FUNCTION_BLOCK _Array0to10OfBool_TestSuite EXTENDS TcUnit.FB_TestSuite
VAR
END_VAR

TestAddress();
TestBaseDatatype();
TestClearReference();
TestClone();
TestGetElementByIndex();
TestTypeNameReturnsExpected();
TestIdentifierReturnsExpected();
TestLength();
TestLowerBound();
TestMakeReferenceToFollowsReference();
TestMakeReferenceToUpdatesReference();
TestSize();
TestSerializeTypeWith();
TestSerializeWith();
TestTryDeserializeFrom();
TestTryMakeReferenceToFollowsReference();
TestTryMakeReferenceToUpdatesReference();
TestUpperBound();
TestValueReturnsExpectedAfterChange();

METHOD PUBLIC TestAddress
VAR
    _type : _Array0to10OfBool;
    notExpected : PVOID := 0;
    actual : PVOID;
END_VAR
TEST('TestAddress');

actual := _type.Address;

AssertFalse(
    Condition := (notExpected = actual),
    Message := 'Type did not return a valid address.'
);

TEST_FINISHED();
END_METHOD

METHOD PUBLIC TestBaseDatatype
VAR
    _type : _Array0to10OfBool;
    expected : T_MAXSTRING := 'BOOL';
    actual : T_MAXSTRING;
END_VAR
TEST('TestBaseDatatype');

actual := _type.BaseDatatype.TypeName;

AssertEquals_STRING(
    Expected := expected,
    Actual := actual,
    Message := 'Type did not return the correct base type'
);

TEST_FINISHED();
END_METHOD

METHOD PUBLIC TestClearReference
VAR
    _type : _Array0to10OfBool;
	target : ARRAY [0..10] OF BOOL;
    expected : ARRAY [0..10] OF BOOL := [FALSE,FALSE,FALSE,FALSE,FALSE,FALSE,FALSE,FALSE,FALSE,FALSE,FALSE];
    actual : ARRAY [0..10] OF BOOL;
END_VAR
TEST('TestClearReference');

_type.MakeReferenceTo(target);
_type.ClearReference();
target[5] := TRUE;

actual := _type.Value;

AssertEquals(
    Expected := expected,
    Actual := actual,
    Message := 'Value incorrectly followed target change'
);

TEST_FINISHED();
END_METHOD

METHOD PUBLIC TestClone
VAR
    _type : _Array0to10OfBool;
	clone : I_Datatype;
	isValidClone : BOOL;
	compareResult : DINT;
END_VAR
TEST('TestClone');

clone := _type.Clone();

isValidClone := clone <> 0;

IF isValidClone THEN
	compareResult := memcmp(_type.Address, clone.Address, clone.Size);
END_IF

AssertTrue(
	Condition := isValidClone,
	Message := 'Clone did not produce a clone'
);

AssertEquals_DINT(
	Expected := 0,
    Actual := compareResult,
    Message := 'Clone did not return a valid clone.'
);

clone.Dispose();

TEST_FINISHED();
END_METHOD

METHOD PUBLIC TestGetElementByIndex
VAR
	_type : _Array0to10OfBool;
    expected : ARRAY [0..10] OF BOOL := [FALSE,FALSE,FALSE,FALSE,FALSE,TRUE,FALSE,FALSE,FALSE,FALSE,FALSE];
    actual : ARRAY [0..10] OF BOOL;
END_VAR
TEST('TestGetElementByIndex');

_type.GetElementByIndex(5).Value := TRUE;

actual := _type.Value;

AssertEquals(
    Expected := expected,
    Actual := actual,
    Message := 'Value did not update target'
);

TEST_FINISHED();
END_METHOD

METHOD PUBLIC TestIdentifierReturnsExpected
VAR
    _type : _Array0to10OfBool;
    expected : STRING := 'ARRAY [0..10] OF BOOL';
    actual : STRING;
END_VAR
TEST('TestIdentifierReturnsExpected');

actual := _type.Identifier;

AssertEquals_STRING(
    Expected := expected,
    Actual := actual,
    Message := 'Type did not return correct iec type.'
);

TEST_FINISHED();
END_METHOD

METHOD PUBLIC TestLength
VAR
    _type : _Array0to10OfBool;
    expected : UDINT := 11;
    actual : UDINT;
END_VAR
TEST('TestLength');

actual := _type.Length;

AssertEquals_UDINT(
    Expected := Expected,
    Actual := actual,
    Message := 'Type did not return the correct array length.'
);

TEST_FINISHED();
END_METHOD

METHOD PUBLIC TestLowerBound
VAR
    _type : _Array0to10OfBool;
    expected : DINT := 0;
    actual : DINT;
END_VAR
TEST('TestLowerBound');

actual := _type.LowerBound;

AssertEquals_DINT(
    Expected := Expected,
    Actual := actual,
    Message := 'Type did not return the correct array lower bound.'
);

TEST_FINISHED();
END_METHOD

METHOD PUBLIC TestMakeReferenceToFollowsReference
VAR
	_type : _Array0to10OfBool;
	target : ARRAY [0..10] OF BOOL;
    expected : ARRAY [0..10] OF BOOL := [TRUE,FALSE,TRUE,FALSE,TRUE,FALSE,TRUE,FALSE,TRUE,FALSE,TRUE];
    actual : ARRAY [0..10] OF BOOL;
END_VAR
TEST('TestMakeReferenceToFollowsReference');

_type.MakeReferenceTo(target);
target[0] := TRUE;
target[2] := TRUE;
target[4] := TRUE;
target[6] := TRUE;
target[8] := TRUE;
target[10] := TRUE;

actual := _type.Value;

AssertEquals(
    Expected := expected,
    Actual := actual,
    Message := 'Value did not follow target change'
);

TEST_FINISHED();
END_METHOD

METHOD PUBLIC TestMakeReferenceToUpdatesReference
VAR
	_type : _Array0to10OfBool;
	target : ARRAY [0..10] OF BOOL;
    expected : ARRAY [0..10] OF BOOL := [TRUE,FALSE,TRUE,FALSE,TRUE,FALSE,TRUE,FALSE,TRUE,FALSE,TRUE];
    actual : ARRAY [0..10] OF BOOL;
END_VAR
TEST('TestMakeReferenceToUpdatesReference');

_type.MakeReferenceTo(target);
_type.Value[0] := TRUE;
_type.Value[2] := TRUE;
_type.Value[4] := TRUE;
_type.Value[6] := TRUE;
_type.Value[8] := TRUE;
_type.Value[10] := TRUE;

actual := target;

AssertEquals(
    Expected := expected,
    Actual := actual,
    Message := 'Value did not update target'
);

TEST_FINISHED();
END_METHOD

METHOD PUBLIC TestSerializeTypeWith
VAR
    _type : _Array0to10OfBool;
    serializer : JsonSerializer;
    expected : STRING(1000) := '{"typeName":"ARRAY","identifier":"ARRAY [0..10] OF BOOL","baseType":{"typeName":"BOOL"}}';
    actual : STRING(1000);
END_VAR
TEST('TestSerializeTypeWith');

serializer.Reset();
_type.SerializeTypeWith(serializer);
serializer.TryGetSerializedData(ADR(actual), SIZEOF(actual));

AssertEquals_STRING(
    Expected := expected,
    Actual := actual,
    Message := 'Serialization of type did not return correct string.'
);

TEST_FINISHED();
END_METHOD

METHOD PUBLIC TestSerializeWith
VAR
    _type : _Array0to10OfBool;
    serializer : JsonSerializer;
    expected : STRING(500) := '[true,false,true,false,true,false,true,false,true,false,true]';
    actual : STRING(500);
END_VAR
TEST('TestSerializeWith');

_type.Value[0] := TRUE;
_type.Value[2] := TRUE;
_type.Value[4] := TRUE;
_type.Value[6] := TRUE;
_type.Value[8] := TRUE;
_type.Value[10] := TRUE;

serializer.Reset();
_type.SerializeWith(serializer);
serializer.TryGetSerializedData(ADR(actual), SIZEOF(actual));

AssertEquals_STRING(
    Expected := expected,
    Actual := actual,
    Message := 'Serialization of type data did not return correct string.'
);

TEST_FINISHED();
END_METHOD

METHOD PUBLIC TestSize
VAR
    _type : _Array0to10OfBool;
	example : ARRAY [0..10] OF BOOL;
    expected : UDINT := SIZEOF(example);
    actual : UDINT;
END_VAR
TEST('TestSize');

actual := _type.Size;

AssertEquals_UDINT(
    Expected := Expected,
    Actual := actual,
    Message := 'Type did not return the correct size.'
);

TEST_FINISHED();
END_METHOD

METHOD PUBLIC TestTryDeserializeFrom
VAR
    deserializer : JsonDeserializer;
    feedback : DeserializerFeedback;
    json : STRING(500) := '[true,false,true,false,true,false,true,false,true,false,true]';
    _type : _Array0to10OfBool;
    expected :  ARRAY [0..10] OF BOOL := [TRUE,FALSE,TRUE,FALSE,TRUE,FALSE,TRUE,FALSE,TRUE,FALSE,TRUE];
    actual : ARRAY [0..10] OF BOOL;
 END_VAR
TEST('TestTryDeserializeFrom');

deserializer.Reset();
deserializer.TryLoad(json);
_type.TryDeserializeFrom(Deserializer, Feedback);

actual := _type.Value;

AssertEquals(
    Expected := expected,
    Actual := actual,
    Message := 'Type did not deserialize correctly.'
);

TEST_FINISHED();
END_METHOD

METHOD PUBLIC TestTryMakeReferenceToFollowsReference
VAR
    _type : _Array0to10OfBool;
	target : _Array0to10OfBool;
    expected : ARRAY [0..10] OF BOOL := [TRUE,FALSE,TRUE,FALSE,TRUE,FALSE,TRUE,FALSE,TRUE,FALSE,TRUE];
    actual :  ARRAY [0..10] OF BOOL;
END_VAR
TEST('TestTryMakeReferenceToFollowsReference');

_type.TryMakeReferenceTo(target);
target.Value[0] := TRUE;
target.Value[2] := TRUE;
target.Value[4] := TRUE;
target.Value[6] := TRUE;
target.Value[8] := TRUE;
target.Value[10] := TRUE;

actual := _type.Value;

AssertEquals(
    Expected := expected,
    Actual := actual,
    Message := 'Value did not follow target change'
);

TEST_FINISHED();
END_METHOD

METHOD PUBLIC TestTryMakeReferenceToUpdatesReference
VAR
    _type : _Array0to10OfBool;
	target : _Array0to10OfBool;
    expected : ARRAY [0..10] OF BOOL := [TRUE,FALSE,TRUE,FALSE,TRUE,FALSE,TRUE,FALSE,TRUE,FALSE,TRUE];
    actual :  ARRAY [0..10] OF BOOL;
END_VAR
TEST('TestTryMakeReferenceToUpdatesReference');

_type.TryMakeReferenceTo(target);
_type.Value[0] := TRUE;
_type.Value[2] := TRUE;
_type.Value[4] := TRUE;
_type.Value[6] := TRUE;
_type.Value[8] := TRUE;
_type.Value[10] := TRUE;

actual := target.Value;

AssertEquals(
    Expected := expected,
    Actual := actual,
    Message := 'Value did not update target'
);

TEST_FINISHED();
END_METHOD

METHOD PUBLIC TestTypeNameReturnsExpected
VAR
    _type : _Array0to10OfBool;
    expected : STRING := 'ARRAY';
    actual : STRING;
END_VAR
TEST('TestTypeNameReturnsExpected');

actual := _type.TypeName;

AssertEquals_STRING(
    Expected := expected,
    Actual := actual,
    Message := 'Type did not return correct iec type.'
);

TEST_FINISHED();
END_METHOD

METHOD PUBLIC TestUpperBound
VAR
    _type : _Array0to10OfBool;
    expected : DINT := 10;
    actual : DINT;
END_VAR
TEST('TestUpperBound');

actual := _type.UpperBound;

AssertEquals_DINT(
    Expected := Expected,
    Actual := actual,
    Message := 'Type did not return the correct array upper bound.'
);

TEST_FINISHED();
END_METHOD

METHOD PUBLIC TestValueReturnsExpectedAfterChange
VAR
    _type : _Array0to10OfBool;
	value : ARRAY [0..10] OF BOOL := [TRUE,FALSE,TRUE,FALSE,TRUE,FALSE,TRUE,FALSE,TRUE,FALSE,TRUE];
    expected : ARRAY [0..10] OF BOOL := [TRUE,FALSE,TRUE,FALSE,TRUE,FALSE,TRUE,FALSE,TRUE,FALSE,TRUE];
    actual :  ARRAY [0..10] OF BOOL;
END_VAR
TEST('TestValueReturnsExpectedAfterChange');

_type.Value := value;
actual := _type.Value;

AssertEquals(
    Expected := expected,
    Actual := actual,
    Message := 'Expected value not returned after change.'
);

TEST_FINISHED();
END_METHOD

END_FUNCTION_BLOCK

(* stored: Version 1.1.0.1, ProductVersion 3.1.4024.13
   POU _Array0to10OfBool_TestSuite: Id {05ba40c9-cdd5-0f8e-1137-4e9b945dc077}, SpecialFunc None
   Method TestAddress: Id {4c6f4390-e020-0a57-35f5-eac1a48edeb9}
   Method TestBaseDatatype: Id {ce9623ba-b86a-001b-1227-f84fa940cb33}
   Method TestClearReference: Id {277eac09-54b3-0555-3c11-8026c32ce5c6}
   Method TestClone: Id {ae46656a-2142-0e4f-066c-7b49090b1db0}
   Method TestGetElementByIndex: Id {9b59ab1b-a862-0761-0817-d3ff4ff618b0}
   Method TestIdentifierReturnsExpected: Id {f4097b4c-437a-0d86-345f-93f4bd5ce951}
   Method TestLength: Id {cebb67d8-c7a3-024a-0f89-dc308f18a3bc}
   Method TestLowerBound: Id {c3c3f8c8-b00f-052d-3b96-487950b5518b}
   Method TestMakeReferenceToFollowsReference: Id {c4c12024-f79e-0f74-3177-16ca551f0b80}
   Method TestMakeReferenceToUpdatesReference: Id {d52d9123-689d-088a-22f6-bf1a7d26d30c}
   Method TestSerializeTypeWith: Id {cc0f2ee7-fd7d-01b6-08b8-2534cee739b1}
   Method TestSerializeWith: Id {aa9aada2-ca55-0625-27ce-ff1fdc792382}
   Method TestSize: Id {2ae6e4ea-0dc6-0e35-242a-128db220e92b}
   Method TestTryDeserializeFrom: Id {df0f8af9-9b82-00ab-0b48-deb06b3f74ed}
   Method TestTryMakeReferenceToFollowsReference: Id {d862a3e0-0629-0dcf-253f-06d7e8e656a2}
   Method TestTryMakeReferenceToUpdatesReference: Id {6e3cf2e8-6568-0978-03de-d6073a349a38}
   Method TestTypeNameReturnsExpected: Id {32b974d8-579f-005a-2524-247e7a7d5678}
   Method TestUpperBound: Id {2a9ebbde-3f34-03fe-102b-f3337322cf3a}
   Method TestValueReturnsExpectedAfterChange: Id {bc3d81e0-34ab-0a32-19fc-69b84d3392cc} *)
